(* Schneider Machine Expert - Basic project es2_2pompe_2max_3soglie_livello_perc, file version 3.0.0.0 *)
(* ProjectInformations: Name=New project *)

HARDWARE
  Cpu 0: TM221C40R
  ModuleExtensionObject 0: TM3AI8/G
  EthernetConfiguration: NetworkName=M221, IpAllocationMode=FixedAddress, IpAddress=0.0.0.0, SubnetMask=0.0.0.0
  SerialLineConfiguration: Baud=Baud19200, Parity=ParityEven, DataBits=DataBits8, StopBits=StopBits1, PhysicalMedium=PhysicalMediumRs485, TransmissionMode=TransmissionModeModbusRtu, SlaveId=1, Addressing=SlaveAddressing
  MastTask: UsePeriodScanMode=false, PeriodScan=100
  FastTask: Period=255
  CpuBehavior: StartingMode=StartAsPreviousState, AutoSaveRamOnEeprom=true, WatchdogPeriod=250

SYMBOLS  (address, symbol, comment, settings)
  %M0       P1_USABILE
  %M1       P2_USABILE
  %M2       PASSATO_SOGLIA_MIN  "Il livello acqua è passato sotto la soglia minima?"
  %M3       PASSATO_SOGLIA_MAX1  "Il livello acqua è passato sopra la soglia 1 massima?"
  %M4       PASSATO_SOGLIA_MAX2  "Il livello acqua è passato sopra la soglia 2 massima?"
  %MD0      LVL_PERC  "Livello acqua percentuale."
  %KD0      MIN_SCALA_GREZZO  [Value=1310724000]
  %KD1      MAX_SCALA_GREZZO  [Value=20000]
  %I0.0     P1_AUTO
  %I0.1     P1_MOTO
  %I0.2     P1_ANOMALIA
  %I0.3     P2_AUTO
  %I0.4     P2_MOTO
  %I0.5     P2_ANOMALIA
  %Q0.0     P1_CMD
  %Q0.1     P2_CMD
  %IW0.0      "Livello acqua (grezzo)."  [Type=Type_0_10V, Scope=Scope_Normal, Minimum=0, Maximum=1000]
  %IW1.0    LVL_INPUT_GREZZO  [Type=Type_4_20mA, Scope=Scope_Customized, Minimum=4000, Maximum=20000]
  %IW1.1    SOGLIA_MIN_PERC  [Type=Type_0_10V, Scope=Scope_Customized, Minimum=0, Maximum=100]
  %IW1.2    SOGLIA_MAX1_PERC  [Type=Type_0_10V, Scope=Scope_Customized, Minimum=0, Maximum=100]
  %IW1.3    SOGLIA_MAX2_PERC  [Type=Type_0_10V, Scope=Scope_Customized, Minimum=0, Maximum=100]

POU Main
  (* SectionNumber=1 *)

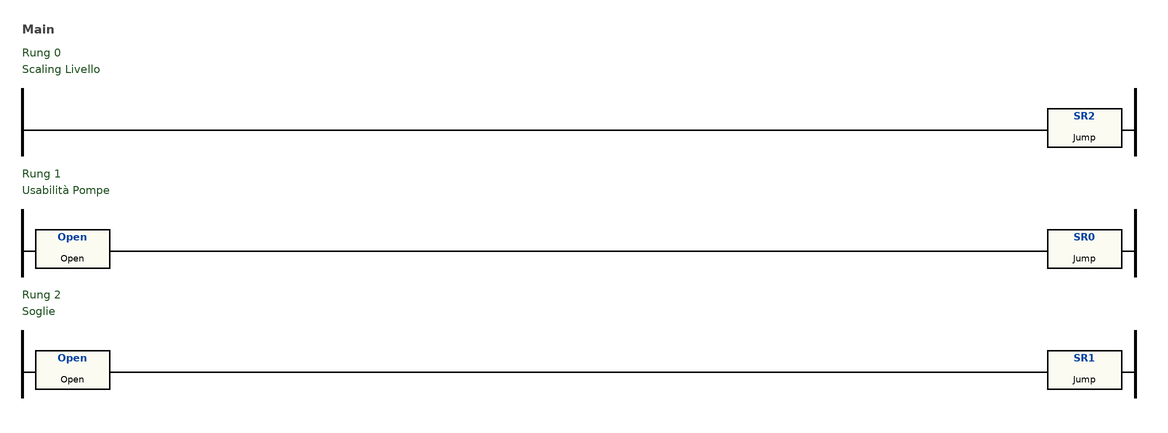

// Rung 0
// Scaling Livello
  LD 1
  SR2
  // as ST:
  //   SR2();

// Rung 1
// Usabilità Pompe
  LD 0
  SR0
  // as ST:
  //   IF FALSE THEN SR0(); END_IF;

// Rung 2
// Soglie
  LD 0
  SR1
  // as ST:
  //   IF FALSE THEN SR1(); END_IF;

Subroutine Usabilità Pompe
  (* SectionNumber=2, Number=0 *)

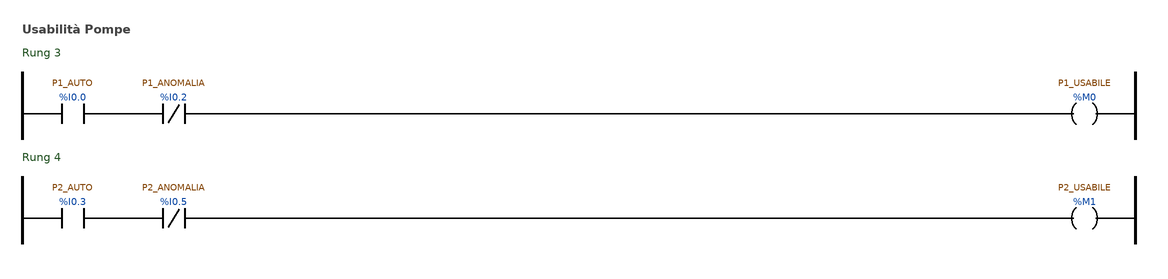

// Rung 3
  LD %I0.0                (* P1_AUTO *)
  ANDN %I0.2              (* P1_ANOMALIA *)
  ST %M0                  (* P1_USABILE *)
  // as ST:
  //   P1_USABILE := P1_AUTO AND NOT P1_ANOMALIA;

// Rung 4
  LD %I0.3                (* P2_AUTO *)
  ANDN %I0.5              (* P2_ANOMALIA *)
  ST %M1                  (* P2_USABILE *)
  // as ST:
  //   P2_USABILE := P2_AUTO AND NOT P2_ANOMALIA;

Subroutine Soglie
  (* SectionNumber=3, Number=1 *)

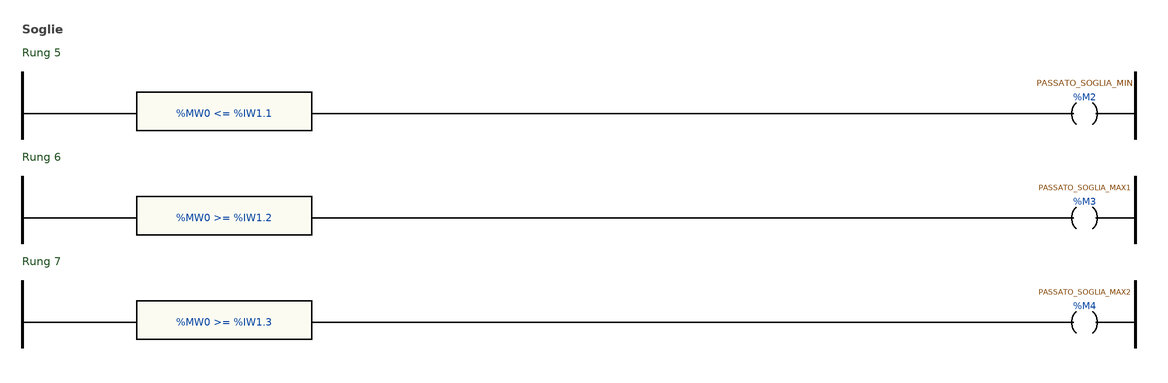

// Rung 5
  LD [ %MW0 <= %IW1.1 ]   (* SOGLIA_MIN_PERC *)
  ST %M2                  (* PASSATO_SOGLIA_MIN *)
  // as ST:
  //   PASSATO_SOGLIA_MIN := %MW0 <= SOGLIA_MIN_PERC;

// Rung 6
  LD [ %MW0 >= %IW1.2 ]   (* SOGLIA_MAX1_PERC *)
  ST %M3                  (* PASSATO_SOGLIA_MAX1 *)
  // as ST:
  //   PASSATO_SOGLIA_MAX1 := %MW0 >= SOGLIA_MAX1_PERC;

// Rung 7
  LD [ %MW0 >= %IW1.3 ]   (* SOGLIA_MAX2_PERC *)
  ST %M4                  (* PASSATO_SOGLIA_MAX2 *)
  // as ST:
  //   PASSATO_SOGLIA_MAX2 := %MW0 >= SOGLIA_MAX2_PERC;

Subroutine Scaling Livello
  (* SectionNumber=4, Number=2 *)

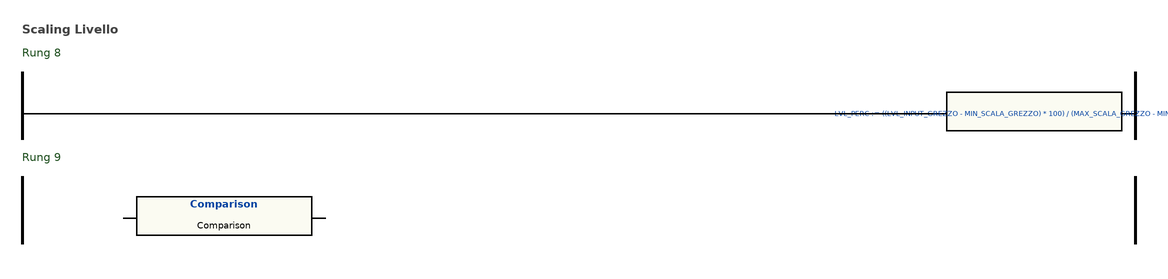

// Rung 8
  (* no IL stored for this rung *)

// Rung 9
  (* no IL stored for this rung *)
